TYPE ST_ItemPK1_OUT2 :
STRUCT
	Identity		:ST_Identity_PK1_OUT2;
	ItemState		:STRING;
	RejectReason	:ST_RejectReason_PK1_OUT2;
	logs			:ST_logs_PK1_OUT2;
	NoRead			:STRING;
END_STRUCT
END_TYPE

(* stored: Version 1.1.0.1, ProductVersion 3.1.4024.13
   DUT ST_ItemPK1_OUT2: Id {e2328124-fa18-4195-b34f-e36b72a61510} *)
